FUNCTION_BLOCK Encoder_Alignment
VAR_INPUT
	NodeID			: BYTE; (* This Port No. addresses the CANopen Node (see System Manager) *)
	Start 			: BOOL;
	Current_State 	: E_Statemachine_State;	
	Statusword		: WORD;	
END_VAR
VAR_OUTPUT
	Controlword 	: WORD;
	Encoder_offset	: WORD;
	Finished		: BOOL;
END_VAR
VAR
	Index 			: BYTE := 0;
	
	SDO_WRITE		: FB_SDO_WRITE;
	WriteData		: ARRAY [0..255] OF BYTE;
	
	SDO_READ		: FB_SDO_READ;
	ReadStart		: BOOL;
	ReadError		: DWORD;
	ReadData		: ARRAY [0..255] OF BYTE;
	
	fbTonDelay		: TON;
	Start_old		: BOOL := FALSE;
END_VAR

// Restart after complete run
IF NOT Start_old AND Start THEN
	Index := 0;
	Finished := FALSE;
END_IF


CASE Index OF	
	0: // Switch to state 'Switch on disabled'
		IF (Start) THEN
			Controlword := CONTROLWORD_STATE_CHANGE(Current_State, E_Statemachine_State.Switch_on_disabled);
			IF (Current_State = E_Statemachine_State.Switch_on_disabled) THEN			
				Index := Index + 2;
			ELSE
				Index := Index + 1;		
			END_IF
		END_IF
		
			
	1: // Wait for 'Switch on disabled'
		Controlword := CONTROLWORD_STATE_CHANGE(Current_State, E_Statemachine_State.Switch_on_disabled);	
		IF (Current_State = E_Statemachine_State.Switch_on_disabled) THEN			
			Index := Index + 1;		
		END_IF
					
		
	2: // Set Mode of operation
		PDO.Mode_of_operation := E_Mode_of_operation.Phasing_mode;	
		Controlword := CONTROLWORD_STATE_CHANGE(Current_State, E_Statemachine_State.Switch_on_disabled);				
		IF (PDO.Mode_of_operation_display = E_Mode_of_operation.Phasing_mode) THEN			
			Index := Index + 1;		
		END_IF

		
	3: // Start
		Controlword := CONTROLWORD_STATE_CHANGE(Current_State, E_Statemachine_State.Operation_enabled);	
		IF ((Current_State = E_Statemachine_State.Operation_enabled) AND ((Statusword AND E_Statusword_Bits.Manufacturer_specific_3) <> 0)) THEN			
			Index := Index + 1;		
		END_IF
		
		
	4: // Wait for finish
		Controlword := CONTROLWORD_STATE_CHANGE(Current_State, E_Statemachine_State.Operation_enabled);			
		IF ((Statusword AND E_Statusword_Bits.Manufacturer_specific_3) = 0) THEN			
			Index := Index + 1;		
		END_IF
	
		
	5: // Switch State to 'Switch on disabled'
		Controlword := CONTROLWORD_STATE_CHANGE(Current_State, E_Statemachine_State.Switch_on_disabled);	
		IF (Current_State = E_Statemachine_State.Switch_on_disabled) THEN			
			Index := Index + 1;
		END_IF
		
		
	6: // Save		
		Controlword := CONTROLWORD_STATE_CHANGE(Current_State, E_Statemachine_State.Switch_on_disabled);	
		WriteData[0] := 16#73;	// s
		WriteData[1] := 16#61;	// a
		WriteData[2] := 16#76;	// v
		WriteData[3] := 16#65;	// e		
		SDO_WRITE(	
			AdsNetID		:= '5.156.6.243.3.1',
			PortNr			:= 16#1000 + NodeID,
			CO_Index		:= 16#1010,
			CO_SubIndex		:= 16#04,
			DataLength		:= 4,
			WriteData		:= WriteData,
			StartWriting	:= TRUE	
		);	
		Index := Index + 1;		

		
	7: // Wait for finish sdo transfer	
		Controlword := CONTROLWORD_STATE_CHANGE(Current_State, E_Statemachine_State.Switch_on_disabled);	
		SDO_WRITE(StartWriting := FALSE);
		IF SDO_WRITE.WriteDataFinished THEN
			Index := Index + 1;			
		END_IF		
		
		
	8: // Wait 500 ms for save process
		Controlword := CONTROLWORD_STATE_CHANGE(Current_State, E_Statemachine_State.Switch_on_disabled);	
		fbTonDelay(IN := TRUE, PT:= T#500MS);
		IF fbTonDelay.Q THEN
			fbTonDelay(IN := FALSE);
			Index := Index + 1;	
		END_IF
		
		
	9: // Read the alignment offset
		Controlword := CONTROLWORD_STATE_CHANGE(Current_State, E_Statemachine_State.Switch_on_disabled);	
		SDO_READ(	
			AdsNetID		:= '5.156.6.243.3.1',
			PortNr			:= 16#1000 + NodeID,
			CO_Index		:= 16#41C0,
			CO_SubIndex		:= 16#11,
			DataLength		:= 2,
			StartReading	:= TRUE	
		);	
		Index := Index + 1;	
		
		
	10: // Wait for finish sdo transfer
		Controlword := CONTROLWORD_STATE_CHANGE(Current_State, E_Statemachine_State.Switch_on_disabled);	
		SDO_Read(StartReading := FALSE);
		IF SDO_WRITE.WriteDataFinished THEN			
			Encoder_offset := SHL(BYTE_TO_WORD(SDO_READ.ReadData[1]),8) + BYTE_TO_WORD(SDO_READ.ReadData[0]);
			Index := 255;			
		END_IF	
			
		
	255: // Finished 
		Controlword := CONTROLWORD_STATE_CHANGE(Current_State, E_Statemachine_State.Switch_on_disabled);	
		FINISHED := TRUE;
				
		
	ELSE
		Index := 255;
			
END_CASE


Start_old := Start;

END_FUNCTION_BLOCK

(* stored: Version 1.1.0.1, ProductVersion 3.1.4024.11
   POU Encoder_Alignment: Id {fffc2c42-72de-4382-ac9e-13e5655c61af}, SpecialFunc None *)
